FUNCTION_BLOCK Phase (* CAT Function Block Type *)
  (* Standard: 61499-2 *)
  (* Version 0.0, 6/4/2026, Schneider Electric, template *)
  PACKAGE SE.Nereda;
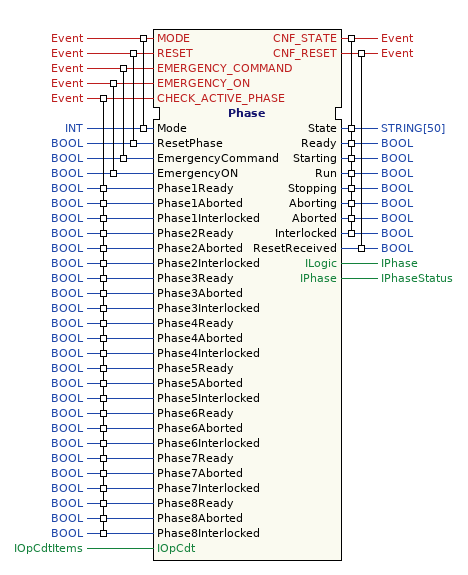
  EVENT_INPUT
    MODE WITH Mode; (* Normal Execution Request *)
    RESET WITH ResetPhase;
    EMERGENCY_COMMAND WITH EmergencyCommand; (* Request for update of status *)
    EMERGENCY_ON WITH EmergencyON; (* Normal Execution Request *)
    CHECK_ACTIVE_PHASE WITH Phase1Ready, Phase1Aborted, Phase1Interlocked, Phase2Ready, Phase2Aborted, Phase2Interlocked, Phase3Ready, Phase3Aborted, Phase3Interlocked, Phase4Ready, Phase4Aborted, Phase4Interlocked, Phase5Ready, Phase5Aborted, Phase5Interlocked, Phase6Ready, Phase6Aborted, Phase6Interlocked, Phase7Ready, Phase7Aborted, Phase7Interlocked, Phase8Ready, Phase8Aborted, Phase8Interlocked; (* Normal Execution Request *)
  END_EVENT
  EVENT_OUTPUT
    CNF_STATE WITH State, Starting, Run, Stopping, Aborting, Aborted, Interlocked, Ready;
    CNF_RESET WITH ResetReceived; (* Execution Confirmation *)
  END_EVENT
  VAR_INPUT
    Mode : INT; (* Argument *)
    ResetPhase : BOOL;
    EmergencyCommand : BOOL; (* Argument *)
    EmergencyON : BOOL; (* Argument *)
    Phase1Ready : BOOL := TRUE; (* Input event qualifier *)
    Phase1Aborted : BOOL := FALSE;
    Phase1Interlocked : BOOL := FALSE; (* Input event qualifier *)
    Phase2Ready : BOOL := TRUE; (* Input event qualifier *)
    Phase2Aborted : BOOL := FALSE;
    Phase2Interlocked : BOOL := FALSE; (* Input event qualifier *)
    Phase3Ready : BOOL := TRUE; (* Input event qualifier *)
    Phase3Aborted : BOOL := FALSE;
    Phase3Interlocked : BOOL := FALSE; (* Input event qualifier *)
    Phase4Ready : BOOL := TRUE; (* Input event qualifier *)
    Phase4Aborted : BOOL := FALSE;
    Phase4Interlocked : BOOL := FALSE; (* Input event qualifier *)
    Phase5Ready : BOOL := TRUE; (* Input event qualifier *)
    Phase5Aborted : BOOL := FALSE;
    Phase5Interlocked : BOOL := FALSE; (* Input event qualifier *)
    Phase6Ready : BOOL := TRUE; (* Input event qualifier *)
    Phase6Aborted : BOOL := FALSE;
    Phase6Interlocked : BOOL := FALSE; (* Input event qualifier *)
    Phase7Ready : BOOL := TRUE; (* Input event qualifier *)
    Phase7Aborted : BOOL := FALSE;
    Phase7Interlocked : BOOL := FALSE; (* Input event qualifier *)
    Phase8Ready : BOOL := TRUE; (* Input event qualifier *)
    Phase8Aborted : BOOL := FALSE;
    Phase8Interlocked : BOOL := FALSE; (* Input event qualifier *)
  END_VAR
  VAR_OUTPUT
    State : STRING[50];
    Ready : BOOL;
    Starting : BOOL;
    Run : BOOL;
    Stopping : BOOL;
    Aborting : BOOL;
    Aborted : BOOL;
    Interlocked : BOOL;
    ResetReceived : BOOL; (* Result: IN1 OR IN2 OR ... *)
  END_VAR
  SOCKETS
    IOpCdt : IOpCdtItems;
  END_SOCKETS
  PLUGS
    ILogic : IPhase;
    IPhase : IPhaseStatus;
  END_PLUGS
  (* 01 - FUNCTIONNAL INPUT INTERFACE *)
  (* 00 - INITIALIZATION *)
  (* 05 - LOGIC *)
  (* 06 - HMI INTERFACE *)
  (* 03 - FIELD INTERFACE *)
  (* 02 - FUNCTIONNAL OUTPUT INTERFACE *)
  (* Phase Manager *)
  (* Operating Condition Status *)
  (* Phase Running Duration *)
  (* Active Phase *)
  (* Name Generator *)
  (* Reset Force Trs *)
  (* State Memo *)
  (* Name Generator *)
  (* Memorize OC *)
  FBS
    Command : Phase_HMI(QI := TRUE);
    INIT : plcStart(Prio := 48, Delay := T#0ms);
    PhaseLogic : PhaseBasic;
    Smooth : boolValueChanged; {SET_ATTRIBUTE(Configuration.Component.HideUnusedPorts, )}
    RunningDurationCalc : devMntCalc(TBaseOperationDuration := T#1s, TBaseElapsedDuration := T#1d); {SET_ATTRIBUTE(Configuration.Component.HideUnusedPorts, )}
    ChekActivePhase : CheckActivePhase;
    NameGenerator : VALFORMAT_8708B18B173C5ABA(FORMAT := '%s', VALUE1 := '$${PATH:3,0}'); {SET_ATTRIBUTE(Configuration.GenericFBType.InterfaceParams, Runtime.Standard#I:=1;VALUE${I$}:STRING)}
    ResetTrsDelay : E_DELAY(DT := T#300ms);
    ResetTrs : TriggerNot0;
    StateMemo : PrevCurrState;
    EmergencyStartCmd : AND_88A3DD8EC65DD11C; {SET_ATTRIBUTE(Configuration.GenericFBType.InterfaceParams, Runtime.Standard#CNT:=2;OUT:BOOL)}
    EmergencyStopCmd : OR_88A3DD8EC65DD11C; {SET_ATTRIBUTE(Configuration.GenericFBType.InterfaceParams, Runtime.Standard#CNT:=2;OUT:BOOL)}
    EmergencyOFF : NOT_42C76073DCEB1A7A; {SET_ATTRIBUTE(Configuration.GenericFBType.InterfaceParams, Runtime.Standard#CNT:=1;OUT${CNT$}:BOOL)}
    EmergencyCmdOFF : NOT_42C76073DCEB1A7A; {SET_ATTRIBUTE(Configuration.GenericFBType.InterfaceParams, Runtime.Standard#CNT:=1;OUT${CNT$}:BOOL)}
    MemoOC : MemoOC_D;
    OR1 : OR_550FE6D62F509EB3; {SET_ATTRIBUTE(Configuration.GenericFBType.InterfaceParams, Runtime.Standard#CNT:=3;OUT:BOOL)}
  END_FBS
  EVENT_CONNECTIONS
    RunningDurationCalc.INITO TO MemoOC.7689825C23C7E3C1;
    RunningDurationCalc.INITO TO NameGenerator.REQ;
    INIT.FIRST_INIT TO Command.681DAFAD0250A347;
    INIT.REDO_INIT TO Command.681DAFAD0250A347;
    NameGenerator.CNF TO Command.AB0DC47F4EE76685;
    RunningDurationCalc.CNF_OPD TO Command.7EE55F02BB0A0EAF;
    MODE TO Command.DBB0F6DA76790C3E;
    ResetTrsDelay.EO TO Command.64D6A61F6AA6E904;
    Command.0AE52BB86A4D3B06 TO RunningDurationCalc.INIT;
    ResetTrsDelay.EO TO Command.0B0477BAA727519B;
    IOpCdt.51FD4CCF54DA16B0 TO Smooth.REQ;
    StateMemo.C79BF2830073106B TO Command.C1FDB87210FE491D;
    StateMemo.C79BF2830073106B TO Command.8776DC5BB4C140DE;
    IOpCdt.0DE1D11A791E8338 TO Command.3B8B0F63AF509F13;
    Command.234A464747DCAA33 TO PhaseLogic.6A6909AB3AC3FE2B;
    Command.234A464747DCAA33 TO ResetTrs.98B4D14610C64DF9;
    Command.3455DE4581509A63 TO PhaseLogic.BC02A417AD186553;
    Command.3455DE4581509A63 TO ResetTrs.98B4D14610C64DF9;
    Command.D4F90E87B63862DD TO PhaseLogic.ED96B16979AE9120;
    Command.D4F90E87B63862DD TO ResetTrs.98B4D14610C64DF9;
    Command.3565A079B3E52930 TO PhaseLogic.C3D98BD2FF4AC1DC;
    Command.E050F8C93EB75AE1 TO PhaseLogic.F80A0F3D9DA66AD6;
    Command.D3A5AE789665DC81 TO PhaseLogic.8506028F5F2CB372;
    Command.2E590CBE9BA06951 TO PhaseLogic.787B96A21DE73C52;
    Command.2E590CBE9BA06951 TO ResetTrs.98B4D14610C64DF9;
    Smooth.CHD TO PhaseLogic.E606389632650A75;
    PhaseLogic.0A98FAF6C5AC2544 TO RunningDurationCalc.REQ_PV;
    PhaseLogic.43A3D11082C8AC90 TO RunningDurationCalc.REQ_RESET;
    ChekActivePhase.CNF TO PhaseLogic.9DC400416FACA09C;
    CHECK_ACTIVE_PHASE TO ChekActivePhase.REQ;
    PhaseLogic.34A75D5169770741 TO StateMemo.0656E54CEB2F117B;
    StateMemo.C79BF2830073106B TO ILogic.Interlocked_CNF;
    StateMemo.C79BF2830073106B TO ILogic.State_CNF;
    StateMemo.C79BF2830073106B TO CNF_STATE;
    StateMemo.C79BF2830073106B TO IPhase.Interlocked_CNF;
    StateMemo.C79BF2830073106B TO IPhase.State_CNF;
    ResetTrs.4D14044435EE07B0 TO ResetTrsDelay.START;
    MODE TO PhaseLogic.FAA67692975EB6BB;
    EMERGENCY_COMMAND TO EmergencyStartCmd.REQ;
    RESET TO PhaseLogic.DF0C6DCA2FCD1007;
    ILogic.REQ_Start_Ready TO PhaseLogic.A1C755A81A4AA94D;
    ILogic.REQ_Stop_Ready TO PhaseLogic.0DD2E2CC19BBF1E2;
    ILogic.REQ_Abort_Ready TO PhaseLogic.5183481590E96066;
    EmergencyStartCmd.CNF TO PhaseLogic.3682FB5FCDD20136;
    EMERGENCY_ON TO EmergencyStartCmd.REQ;
    EmergencyStopCmd.CNF TO PhaseLogic.4C073025D79B7E33;
    EmergencyOFF.CNF TO EmergencyStopCmd.REQ;
    EmergencyCmdOFF.CNF TO EmergencyOFF.REQ;
    EMERGENCY_COMMAND TO EmergencyCmdOFF.REQ;
    EMERGENCY_ON TO EmergencyCmdOFF.REQ;
    MemoOC.E74FDFC5C9E17061 TO INIT.ACK_FIRST;
    IOpCdt.510B9224626AA5DB TO MemoOC.ABF856B2CD45BEB5;
    RESET TO OR1.REQ;
    Command.D3A5AE789665DC81 TO OR1.REQ;
    Command.D4F90E87B63862DD TO OR1.REQ;
    OR1.CNF TO CNF_RESET;
  END_CONNECTIONS
  DATA_CONNECTIONS
    NameGenerator.RESULT TO Command.84AFB794FDC11D00;
    RunningDurationCalc.CurrentOperationDuration TO Command.859517F20FDFEA1E;
    Mode TO Command.DD344CAE687A6888;
    IOpCdt.5E924D1CC4B831CF TO Smooth.Input;
    PhaseLogic.67153EDE3BF57436 TO Command.7FBACF637741D948;
    PhaseLogic.ED7331EB76A66CEF TO Command.63BE7C67CD79D37C;
    PhaseLogic.6BC2EEC4FF5D5F73 TO Command.A82CD0475A5C0310;
    PhaseLogic.CCA1C294F958E66A TO Command.FB5D348A591BEFC9;
    PhaseLogic.B4B0727567B73B53 TO Command.807DEB8EB9CAA816;
    PhaseLogic.C90894D28A9EDEEB TO Command.2D4DA52AB4ED86E0;
    PhaseLogic.20EABBC4E43F76A9 TO Command.C73A321B4927C334;
    PhaseLogic.5788AC25D2ED9221 TO Command.5FF908AC0B069C33;
    PhaseLogic.74960193A135381A TO Command.DA3C45E7DDF926D6;
    StateMemo.EBE08A4AE843EBA3 TO Command.CC116D014291EE77;
    StateMemo.4B6C97D21C93CAE0 TO Command.9ECFB4DCC3962B12;
    IOpCdt.83A3C315F80CFE17 TO Command.ED67C2E6B51A0D30;
    IOpCdt.B50BFE7459784F00 TO Command.0AEA0D2A2340FF57;
    IOpCdt.946A0F582B551978 TO Command.007DBDD0734A6B08;
    IOpCdt.FCEA282DF5077920 TO Command.7ACBE634044AE3F9;
    IOpCdt.2B4F39E9175B3855 TO Command.3CFA3B6969FA8D87;
    IOpCdt.4596A1B27C10C2CD TO Command.6D222C63F400B0EF;
    IOpCdt.A9753615DA8DD82A TO Command.616BCC4FB156170B;
    IOpCdt.824CE9000F3F9466 TO Command.88CD56238581AA36;
    IOpCdt.72067FEC91126715 TO Command.F5EC6C52DDCAEBF2;
    IOpCdt.37C7DD09745BE300 TO Command.1571D6BB1FFADCD4;
    IOpCdt.03CAF86670282F7A TO Command.82CC44B926CB9F7F;
    IOpCdt.A578CCE6834280A9 TO Command.9B5BDFDAB51136DE;
    IOpCdt.932E293892006A0F TO Command.A9D7A4CC6E3A64E2;
    IOpCdt.3136228301C0A3F6 TO Command.7931F46F07FB68CD;
    IOpCdt.BBA5573FBFE93EF1 TO Command.42538CBE9623CA73;
    IOpCdt.9095F08A1259C467 TO Command.4DF68C8A27457CDE;
    IOpCdt.87CAB742E188E408 TO Command.8597C48C2E3C6C5E;
    IOpCdt.315583C88EDCE2AB TO Command.07C68CAB1F60A717;
    IOpCdt.DC6E7346CAD3F412 TO Command.C5128310633CF49C;
    IOpCdt.154499D847362610 TO Command.6AB5F3284A1BA77D;
    Command.F75BBC3D25B9E108 TO PhaseLogic.8F473934F997BE28;
    Command.F75BBC3D25B9E108 TO ResetTrs.29D805626EF42DFD;
    Command.16624A9387C45D3D TO PhaseLogic.6500FD2ED27DE4F8;
    Command.16624A9387C45D3D TO ResetTrs.4C3690459161CE49;
    Command.128886B65D60AE22 TO PhaseLogic.6FA16472453C7E6E;
    Command.128886B65D60AE22 TO ResetTrs.F49257499C4544D7;
    Command.BFBD1A8C7D1A5D7E TO PhaseLogic.ABF982FA0C85D538;
    Command.AA18D73C64A29EA4 TO PhaseLogic.070CE521296D2865;
    Command.CC1A93ACAA9A6147 TO PhaseLogic.165A320E06831D77;
    Command.106B09E4726D073E TO PhaseLogic.877C261E0F9EB68F;
    Command.106B09E4726D073E TO ResetTrs.622EA78CA147C620;
    Smooth.Output TO PhaseLogic.ED9B68DAECDB184C;
    PhaseLogic.976B5CF28484676F TO RunningDurationCalc.Pv;
    PhaseLogic.20DFC8514AB2A821 TO RunningDurationCalc.ResetOperationDuration;
    ChekActivePhase.NoActivePhase TO PhaseLogic.71A2A3118846C5EF;
    Phase4Interlocked TO ChekActivePhase.143EC1F8D1452500;
    Phase4Ready TO ChekActivePhase.5631C79DD3FFB37A;
    Phase3Interlocked TO ChekActivePhase.230F46FBD6471F96;
    Phase3Ready TO ChekActivePhase.IN7;
    Phase2Interlocked TO ChekActivePhase.IN6;
    Phase2Ready TO ChekActivePhase.IN4;
    Phase1Interlocked TO ChekActivePhase.IN3;
    Phase1Ready TO ChekActivePhase.IN1;
    PhaseLogic.74960193A135381A TO StateMemo.8C198C6E6A0624DE;
    Mode TO PhaseLogic.671E31693D4596AA;
    EmergencyCommand TO EmergencyStartCmd.IN1;
    ResetPhase TO PhaseLogic.B44471DB4E020AD1;
    ILogic.Start_Ready TO PhaseLogic.D40CA51700732AA8;
    ILogic.Stop_Ready TO PhaseLogic.0A4B6A57D9914D6D;
    ILogic.Abort_Ready TO PhaseLogic.B8A6E7DE75D7616B;
    PhaseLogic.67153EDE3BF57436 TO ILogic.Ready;
    PhaseLogic.ED7331EB76A66CEF TO ILogic.Starting;
    PhaseLogic.6BC2EEC4FF5D5F73 TO ILogic.Run;
    PhaseLogic.CCA1C294F958E66A TO ILogic.Stopping;
    PhaseLogic.B4B0727567B73B53 TO ILogic.Aborting;
    PhaseLogic.C90894D28A9EDEEB TO ILogic.Aborted;
    PhaseLogic.20EABBC4E43F76A9 TO ILogic.Interlocked;
    PhaseLogic.5788AC25D2ED9221 TO ILogic.State;
    PhaseLogic.67153EDE3BF57436 TO IPhase.Ready;
    PhaseLogic.ED7331EB76A66CEF TO IPhase.Starting;
    PhaseLogic.6BC2EEC4FF5D5F73 TO IPhase.Run;
    PhaseLogic.CCA1C294F958E66A TO IPhase.Stopping;
    PhaseLogic.B4B0727567B73B53 TO IPhase.Aborting;
    PhaseLogic.C90894D28A9EDEEB TO IPhase.Aborted;
    PhaseLogic.20EABBC4E43F76A9 TO IPhase.Interlocked;
    PhaseLogic.5788AC25D2ED9221 TO IPhase.State;
    PhaseLogic.5788AC25D2ED9221 TO State;
    PhaseLogic.67153EDE3BF57436 TO Ready;
    PhaseLogic.ED7331EB76A66CEF TO Starting;
    PhaseLogic.6BC2EEC4FF5D5F73 TO Run;
    PhaseLogic.CCA1C294F958E66A TO Stopping;
    PhaseLogic.B4B0727567B73B53 TO Aborting;
    PhaseLogic.C90894D28A9EDEEB TO Aborted;
    PhaseLogic.20EABBC4E43F76A9 TO Interlocked;
    EmergencyStartCmd.OUT TO PhaseLogic.7CABF06C0A678B59;
    EmergencyON TO EmergencyStartCmd.IN2;
    EmergencyStopCmd.OUT TO PhaseLogic.F7741ED7387A838E;
    EmergencyOFF.OUT1 TO EmergencyStopCmd.IN1;
    EmergencyCommand TO EmergencyCmdOFF.IN1;
    EmergencyON TO EmergencyOFF.IN1;
    EmergencyCmdOFF.OUT1 TO EmergencyStopCmd.IN2;
    Phase1Aborted TO ChekActivePhase.IN2;
    Phase2Aborted TO ChekActivePhase.IN5;
    Phase3Aborted TO ChekActivePhase.IN8;
    Phase4Aborted TO ChekActivePhase.0D8DBF99DEDCAC31;
    IOpCdt.7FD7CF3BAAB2C8B1 TO MemoOC.5F9F4453AA72EEC2;
    Command.CC1A93ACAA9A6147 TO OR1.IN1;
    Command.128886B65D60AE22 TO OR1.IN2;
    ResetPhase TO OR1.IN3;
    OR1.OUT TO ResetReceived;
  END_CONNECTIONS
END_FUNCTION_BLOCK
